Yaskawa INFORM job: AAA.JBI

/JOB
//NAME AAA
//POS
///NPOS 1,0,0,0,0,0
///TOOL 12
///POSTYPE PULSE
///PULSE
C00000=0,0,0,0,0,0
//INST
///DATE 2025/03/18 16:03
///ATTR SC,RW
///GROUP1 RB2
NOP
MOVJ C00000 VJ=1.0 PL=0
TIMER T=5.00
END
